Fanuc TP program (LS listing): SEARCH.LS

/PROG  SEARCH
/ATTR
OWNER		= MNEDITOR;
COMMENT		= "";
PROG_SIZE	= 191;
CREATE		= DATE 80-01-01  TIME 00:38:56;
MODIFIED	= DATE 80-01-01  TIME 00:40:36;
FILE_NAME	= ;
VERSION		= 0;
LINE_COUNT	= 3;
MEMORY_SIZE	= 551;
PROTECT		= READ_WRITE;
TCD:  STACK_SIZE	= 0,
      TASK_PRIORITY	= 50,
      TIME_SLICE	= 0,
      BUSY_LAMP_OFF	= 0,
      ABORT_REQUEST	= 0,
      PAUSE_REQUEST	= 0;
DEFAULT_GROUP	= 1,*,*,*,*;
CONTROL_CODE	= 00000000 00000000;
/APPL
  ARC Welding Equipment : 1,*,*,*,*;
/MN
   1:  SENSOR SEARCH START PR[1:HOME_00] ;
   2:  SENSOR SEARCH POINT[1]    ;
   3:  SENSOR SEARCH END ;
/POS
/END
